// TIA Portal V20 export
DATA_BLOCK "PM03"   // DB338
// stored: MemoryReserve 100
   VAR
      "SEPA CUTTER REAR UP / SEPA CUTTER FRONT UP" : Bool := FALSE;
      "SEPA CUTTER REAR DOWN / SEPA CUTTER FRONT DOWN" : Bool := FALSE;
      "SEPA CLAMP TOP REAR UP" : Bool := FALSE;
      "SEPA CLAMP TOP REAR DOWN" : Bool := FALSE;
      "SEPA CLAMP TOP FRONT UP" : Bool := FALSE;
      "SEPA CLAMP TOP FRONT DOWN" : Bool := FALSE;
      "SEPA CLAMP BTM REAR UP" : Bool := FALSE;
      "SEPA CLAMP BTM REAR DOWN" : Bool := FALSE;
      "SEPA CLAMP BTM FRONT UP" : Bool := FALSE;
      "SEPA CLAMP BTM FRONT DOWN" : Bool := FALSE;
      "SEPA GRIPPER OPEN" : Bool := FALSE;
      "SEPA GRIPPER  CLOSE" : Bool := FALSE;
      "SEPA GRIPPER FORWARD" : Bool := FALSE;
      "SEPA GRIPPER BACKWARD" : Bool := FALSE;
   END_VAR
BEGIN
END_DATA_BLOCK
